(*
SPDX-FileCopyrightText: © 2026 Oleksandr Tiutyk <trofimich@gmail.com>
SPDX-License-Identifier: MIT
License: https://opensource.org/license/mit
*)

(*!
<summary>Defines electrical contact type for digital input and output signals.</summary>
<description>
Determines whether the physical signal state is inverted when mapped to the logical component Value.
NORMALLY_OPEN: logical TRUE matches physical TRUE. NORMALLY_CLOSED: logical TRUE matches physical FALSE
(inverted).
</description>
*)

{attribute 'qualified_only'}
{attribute 'strict'}
{attribute 'to_string'}
TYPE CONTACT_TYPE :
(
	NORMALLY_OPEN := 0,
	NORMALLY_CLOSED := 1
);
END_TYPE

(* stored: Version 1.1.0.1
   DUT CONTACT_TYPE: Id {e627eeef-55fa-4d5f-b071-58620f4fab9c} *)
